Universal Robots PolyScope program: pourAndPutDown3.urp

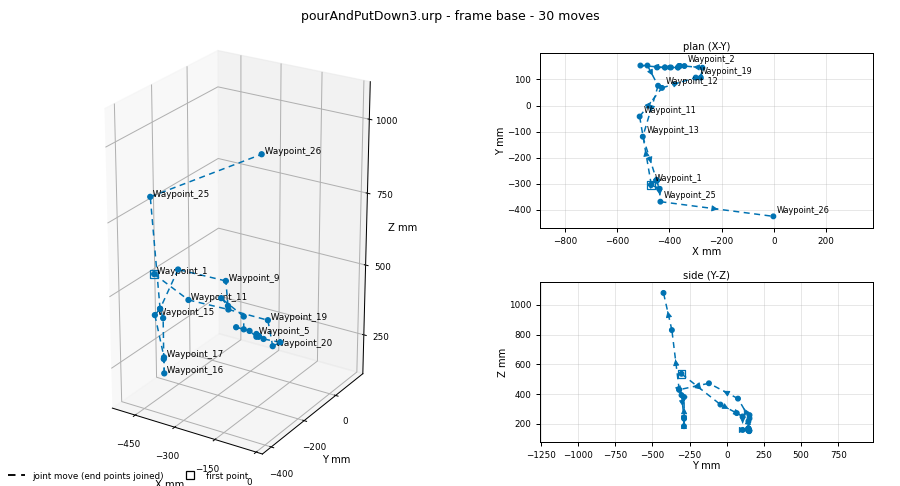
[picture p0: tool path of pourAndPutDown3.urp in frame base, 30 of 30 moves have a stored position in this frame; points joined in program order, loops and branches not executed]
Program pourAndPutDown3 (installation=default directory=/programs/PrakjoyShi_Beer createdIn=5.12.6.1102099 lastSavedIn=5.12.6.1102099 robotSerialNumber=20215500597)
Calibrated DH parameters: a=[0.000193, -0.066673, -0.391568, -0.000012, 0.00005, 0]; d=[0.162643, -472.05677, 465.132521, 7.058239, 0.099746, 0.099582]; alpha=[1.571116, 0.00089, 0.003862, 1.569269, -1.569248, 0]; deltaTheta=[0, -1.413394, 7.628392, 0.068187, 0, -0.000001]
Robot Program (runOnlyOnce=true)
  MoveJ speed 60 deg/s, acceleration 80 deg/s^2 (useActiveTCP=true) feature=Base
    Waypoint Waypoint_1: TCP in base x=-469.422 y=-303.772 z=537.049 mm, rx=-0.9663 ry=-1.499 rz=1.6747 rad; joints [6.908, -106.662, 129.097, -206.194, -67.737, 6.591] deg; TCP offset x=0 y=0 z=191.5 mm, rx=0 ry=0 rz=0 rad
    Waypoint Waypoint_11: TCP in base x=-514.044 y=-42.229 z=330.478 mm, rx=0.9483 ry=1.8098 rz=-1.8406 rad; joints [-42.944, -57.453, 101.188, -230.29, 31.853, 49.611] deg
    Waypoint Waypoint_12: TCP in base x=-428.386 y=67.501 z=272.98 mm, rx=0.8234 ry=1.7173 rz=-1.638 rad; joints [-53.416, -47.466, 95.297, -230.558, 54.247, 53.558] deg
    Waypoint Waypoint_19: TCP in base x=-299.055 y=107.007 z=250.481 mm, rx=0.7818 ry=1.7818 rz=-1.7132 rad; joints [-69.052, -50.894, 107.804, -239.624, 68.324, 47.588] deg
    Waypoint Waypoint_20: TCP in base x=-279.734 y=106.984 z=159.803 mm, rx=0.7816 ry=1.7818 rz=-1.7132 rad; joints [-71.245, -40.233, 108.371, -250.83, 70.508, 47.507] deg
    Waypoint Waypoint_21: TCP in base x=-273.429 y=144.767 z=159.8 mm, rx=0.7817 ry=1.7819 rz=-1.7133 rad; joints [-73.337, -38.608, 103.329, -247.386, 72.596, 47.386] deg; TCP offset x=0 y=0 z=191.5 mm, rx=0 ry=0 rz=0 rad
    Waypoint Waypoint_2: TCP in base x=-342.426 y=151.266 z=151.388 mm, rx=0.9523 ry=1.6137 rz=-1.4653 rad; joints [-64.863, -34.688, 92.564, -242.174, 67.302, 65.082] deg; TCP offset x=0 y=0 z=191.5 mm, rx=0 ry=0 rz=0 rad
    Waypoint Waypoint_22: TCP in base x=-361.408 y=151.426 z=156.141 mm, rx=1.2521 ry=1.214 rz=-1.0973 rad; joints [-63.123, -33.882, 90.405, -239.877, 65.554, 95.492] deg
    Waypoint Waypoint_3: TCP in base x=-361.415 y=151.432 z=156.134 mm, rx=1.2971 ry=1.142 rz=-1.0272 rad; joints [-63.122, -33.883, 90.401, -239.879, 65.554, 101] deg; TCP offset x=0 y=0 z=191.5 mm, rx=0 ry=0 rz=0 rad
    Wait Sleep waitTime=4
    Waypoint Waypoint_4: TCP in base x=-361.423 y=151.429 z=156.139 mm, rx=1.3278 ry=1.0892 rz=-0.9759 rad; joints [-63.123, -33.884, 90.403, -239.879, 65.551, 105] deg; TCP offset x=0 y=0 z=191.5 mm, rx=0 ry=0 rz=0 rad
    Wait Sleep waitTime=6
    Waypoint Waypoint_4: TCP in base x=-361.423 y=151.429 z=156.139 mm, rx=1.3278 ry=1.0892 rz=-0.9759 rad; joints [-63.123, -33.884, 90.403, -239.879, 65.551, 105] deg
    Wait Sleep waitTime=6
    Waypoint Waypoint_5: TCP in base x=-367.114 y=145.876 z=165.681 mm, rx=1.0874 ry=1.5479 rz=-1.4306 rad; joints [-64.058, -36.96, 92.743, -241.765, 62.844, 71.518] deg; TCP offset x=0 y=0 z=191.5 mm, rx=0 ry=0 rz=0 rad
    Waypoint Waypoint_6: TCP in base x=-367.056 y=145.739 z=155.514 mm, rx=0.9649 ry=1.7071 rz=-1.5492 rad; joints [-64.055, -36.274, 92.398, -243.123, 62.84, 60.719] deg
    Waypoint Waypoint_7: TCP in base x=-394.155 y=145.769 z=170.181 mm, rx=0.9649 ry=1.707 rz=-1.5494 rad; joints [-61.586, -36.44, 89.13, -239.83, 60.388, 61.045] deg
    Waypoint Waypoint_8: TCP in base x=-447.148 y=145.786 z=170.185 mm, rx=0.9649 ry=1.707 rz=-1.5493 rad; joints [-57.124, -33.176, 81.279, -235.57, 55.977, 61.696] deg
    Waypoint Waypoint_27: TCP in base x=-417.072 y=145.782 z=170.171 mm, rx=0.9649 ry=1.707 rz=-1.5493 rad; joints [-59.594, -35.095, 85.865, -238.047, 58.422, 61.332] deg
    Waypoint Waypoint_28: TCP in base x=-417.06 y=145.793 z=217.836 mm, rx=0.9649 ry=1.7071 rz=-1.5492 rad; joints [-59.599, -39.934, 86.457, -233.799, 58.436, 61.32] deg
    Waypoint Waypoint_10: TCP in base x=-511.018 y=153.193 z=259.457 mm, rx=1.3001 ry=1.2115 rz=-1.0454 rad; joints [-51.404, -33.693, 66.157, -218.964, 54.247, 100.369] deg
    Waypoint Waypoint_29: TCP in base x=-484.137 y=153.178 z=237.569 mm, rx=1.5023 ry=0.815 rz=-0.6758 rad; joints [-53.239, -34.363, 71.466, -223.469, 56.064, 129.133] deg
    Wait Sleep waitTime=2
    Waypoint Waypoint_9: TCP in base x=-443.299 y=75.819 z=370.314 mm, rx=-0.1462 ry=2.1698 rz=-2.071 rad; joints [-49.086, -50.8, 82.87, -214.951, 58.642, 3.159] deg
    Waypoint Waypoint_13: TCP in base x=-501.996 y=-119.391 z=473.346 mm, rx=-0.1865 ry=2.1452 rz=-2.0717 rad; joints [-29.839, -60.518, 82.876, -205.008, 41.125, 3.179] deg
    Waypoint Waypoint_14: TCP in base x=-438.339 y=-319.405 z=430.326 mm, rx=-0.0095 ry=-2.2019 rz=2.1503 rad; joints [-14.551, -76.261, 113.55, -222.987, 11.638, 3.16] deg
    Waypoint Waypoint_15: TCP in base x=-469.43 y=-303.759 z=393.841 mm, rx=-0.9664 ry=-1.499 rz=1.6746 rad; joints [6.93, -89.791, 142.194, -236.128, -67.835, 6.514] deg
    Waypoint Waypoint_17: TCP in base x=-447.918 y=-287.369 z=242.661 mm, rx=-0.8716 ry=-1.6291 rz=1.5246 rad; joints [1.903, -63.887, 152.292, -266.285, -61.848, -4.367] deg
    Waypoint Waypoint_16: TCP in base x=-447.928 y=-287.349 z=184.854 mm, rx=-0.8716 ry=-1.6291 rz=1.5245 rad; joints [1.931, -47.58, 150.654, -280.927, -61.868, -4.426] deg
    URCap Gripper (Robotiq_Grippers, Robotiq Inc.) dataModel(position=0.0, force=100.0, speed=100.0, positionInDouble=0.0, forceInDouble=100.0, speedInDouble=100.0, slaveIds=[9], blocking=true)
    Waypoint Waypoint_23: TCP in base x=-449.756 y=-286.313 z=235.635 mm, rx=-0.8887 ry=-1.6496 rz=1.5115 rad; joints [1.701, -63.9, 152.473, -264.905, -61.738, -4.834] deg
    Waypoint Waypoint_24: TCP in base x=-449.701 y=-286.338 z=380.979 mm, rx=-0.8887 ry=-1.6496 rz=1.5116 rad; joints [1.635, -100.122, 146.36, -222.64, -61.621, -4.69] deg
    Waypoint Waypoint_18: TCP in base x=-438.34 y=-319.404 z=430.315 mm, rx=-0.0095 ry=-2.2019 rz=2.1504 rad; joints [-14.551, -76.26, 113.551, -222.987, 11.638, 3.162] deg
    Waypoint Waypoint_25: TCP in base x=-434.434 y=-368.574 z=830.932 mm, rx=-0.0069 ry=-2.2054 rz=2.1858 rad; joints [-7.724, -82.704, 60.285, -160.607, 6.18, 1.676] deg
    Waypoint Waypoint_26: TCP in base x=-1.558 y=-424.817 z=1080.554 mm, rx=-0.0044 ry=-2.2185 rz=2.2204 rad; joints [-0.002, -89.999, -0.001, -89.999, 0.002, 0] deg
